FUNCTION_BLOCK FB_MatrixDeterminate_Test EXTENDS FB_TestSuite
VAR_INPUT
END_VAR
VAR_OUTPUT
END_VAR
VAR
END_VAR

WhenNotSquareExpectError();
WhenMatchingExpectResult();

METHOD PRIVATE WhenMatchingExpectResult
VAR_INPUT
END_VAR
VAR
	M1 : DynamicMatrix;
	Result : BOOL;
	Actual : LREAL;
	Expected : LREAL := 360;
END_VAR
TEST('WhenMatchingExpectResult');

// @TEST-RUN
M1.InitMagicSquare(3);
Result := Matrix_Determinate(M := M1,Res => Actual);

// @TEST-ASSERT
AssertTrue(Result,'Main function call was not successful');
AssertEquals(Expected,Actual,'Determinate value was incorrect');

TEST_FINISHED();
END_METHOD

METHOD PRIVATE WhenNotSquareExpectError
VAR_INPUT
END_VAR
VAR
	M1 : DynamicMatrix;
	Result : BOOL;
	Actual : LREAL;
	Expected : LREAL := 0;
END_VAR
TEST('WhenNotSquareExpectError');

// @TEST-RUN
M1.InitTrapezoidal(2,3,1,1,1);
Result := Matrix_Determinate(M := M1,Res => Actual);

// @TEST-ASSERT
AssertFalse(Result,'Main function call was unexpectedly successful');
AssertEquals(Expected,Actual,'Determinate value was incorrect');

TEST_FINISHED();
END_METHOD

END_FUNCTION_BLOCK

(* stored: Version 1.1.0.1, ProductVersion 3.1.4024.9
   POU FB_MatrixDeterminate_Test: Id {05d09fac-54aa-03fb-32bc-a7271461908b}, SpecialFunc None
   Method WhenMatchingExpectResult: Id {861ae7e2-3c14-05ef-31e2-8fb2373cafa7}
   Method WhenNotSquareExpectError: Id {47a4dc4c-d738-0f7a-3585-802d49f8721f} *)
